INTERFACE ITF_Group2_HMI_Init EXTENDS ITF_BaseGroupElement, ITF_Group2_HMI_Connector

END_INTERFACE

(* stored: Version 1.1.0.1
   Itf ITF_Group2_HMI_Init: Id {1d02d036-4b9b-0e86-2196-330737631fcf} *)
